(* Logix 5000 project; controller WASH Emulate 5570 rev 33.11; software revision 33.00 *)

TASK MainTask (continuous, watchdog 500 ms) : MainProgram, Model

MODULES
   Local : Emulate 5570 (ICP 2, rev 33.11)
       : 1756-IB16 (ICP 3, rev 3.1, Input RPI 20 ms)
       : vendor 1 type 7 code 16 (ICP 4, rev 3.1, Output RPI 20 ms)
END_MODULES

PROGRAM MainProgram   (* main routine TextRoutine *)

ROUTINE TextRoutine   (* structured text *)
   
   
END_ROUTINE
END_PROGRAM

PROGRAM Model   (* main routine Emulate *)
VAR
   HOLD : DINT;
   SOL_1_CLSD : TIMER := (PRE := 3000);
   SOL_1_OPN : TIMER := (PRE := 1000);
   SOL_2_CLSD : TIMER := (PRE := 1000);
   SOL_2_OPN : TIMER := (PRE := 2000);
END_VAR

ROUTINE Emulate   (* ladder *)
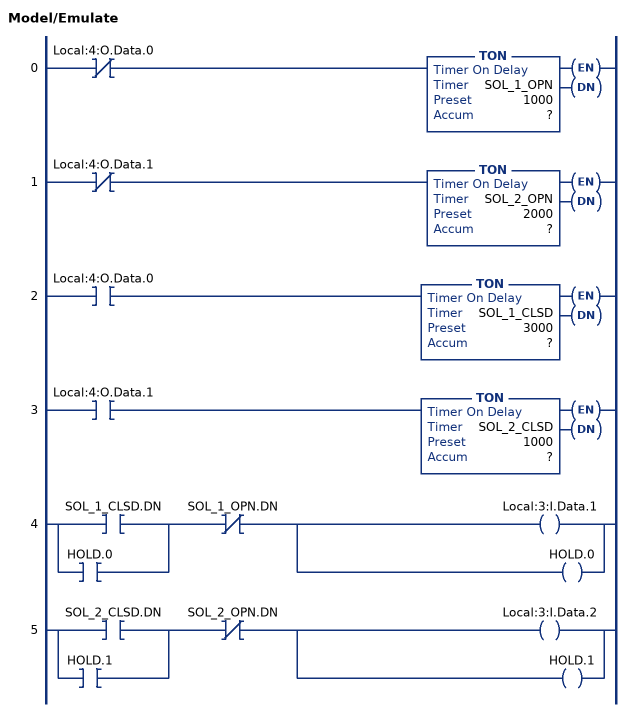
   0: XIO(Local:4:O.Data.0)TON(SOL_1_OPN,?,?);
   1: XIO(Local:4:O.Data.1)TON(SOL_2_OPN,?,?);
   2: XIC(Local:4:O.Data.0)TON(SOL_1_CLSD,?,?);
   3: XIC(Local:4:O.Data.1)TON(SOL_2_CLSD,?,?);
   4: [XIC(SOL_1_CLSD.DN) ,XIC(HOLD.0) ]XIO(SOL_1_OPN.DN)[OTE(Local:3:I.Data.1) ,OTE(HOLD.0) ];
   5: [XIC(SOL_2_CLSD.DN) ,XIC(HOLD.1) ]XIO(SOL_2_OPN.DN)[OTE(Local:3:I.Data.2) ,OTE(HOLD.1) ];
END_ROUTINE
END_PROGRAM
